// TIA Portal V20 export
TYPE "typeCmControlNodeInterlock"
// stored: Namespace Unit1.Em7
   STRUCT
      hotPressRightServoPress : "LER_typeServoPressInterlock";
      hotPressRightStageLiftFront : "LER_typeTwoWayActuatorInterlock";
      hotPressRightStageLiftRear : "LER_typeTwoWayActuatorInterlock";
      hotPressRightStageLiftAll : "LER_typeTwoWayActuatorInterlock";
   END_STRUCT;
END_TYPE
